// TIA Portal V20 export
// export: Created 2026-10-09T07:54:14.9470131Z, ExportSetting WithDefaults, DisplayName Totally Integrated Automation Portal, DisplayVersion V20, DisplayName TIA Portal Openness, DisplayVersion V20, DisplayName TIA Portal Teamcenter Gateway, DisplayVersion V20, DisplayName TIA Portal Version Control Interface, DisplayVersion V20, DisplayName SINAMICS Startdrive Advanced, DisplayVersion V20 SP1 Update 2, DisplayName SINAMICS Startdrive G110M, G120, G120C, G120D, G120P, G115D, DisplayVersion V20 SP1 Update 2, DisplayName SINAMICS Startdrive G130, G150, S120, S150, SINAMICS MV, G220, S200, S210, DisplayVersion V20 SP1 Update 2, DisplayName STEP 7 Professional, DisplayVersion V20, DisplayName STEP 7 Safety, DisplayVersion V20, DisplayName WinCC Basic/Comfort/Advanced, DisplayVersion V20, DisplayName WinCC Professional, DisplayVersion V20, DisplayName WinCC Unified, DisplayVersion V20
FUNCTION_BLOCK "FB_SpkAutoGraph"   // FB30, GRAPH
VERSION : 0.1
// stored: AcknowledgeErrorsRequired true, AutoNumber true, GraphVersion 6.0, InitialValuesAcquisition false, IsIECCheckEnabled false, LanguageInNetworks LAD, LockOperatingMode false, PermanentILProcessingInMANMode false, SetENOAutomatically false, SkipSteps false, UDAEnableTagReadback false, WithAlarmHandling true
   // inherited from GRAPH_BASE
   VAR
      OFF_SQ_BASE : Bool;
   END_VAR
   VAR_INPUT
      OFF_SQ { ExternalAccessible := 'False'; ExternalVisible := 'False'; ExternalWritable := 'False'} : Bool := false;   // Turn sequence off
      INIT_SQ { ExternalAccessible := 'False'; ExternalVisible := 'False'; ExternalWritable := 'False'} : Bool := false;   // Set sequence to initial state
      ACK_EF { ExternalAccessible := 'False'; ExternalVisible := 'False'; ExternalWritable := 'False'} : Bool := false;   // Acknowledge all errors and faults
      S_PREV { ExternalAccessible := 'False'; ExternalVisible := 'False'; ExternalWritable := 'False'} : Bool := false;   // Output previous step in parameter S_NO
      S_NEXT { ExternalAccessible := 'False'; ExternalVisible := 'False'; ExternalWritable := 'False'} : Bool := false;   // Indicate next step in parameter S_NO
      SW_AUTO { ExternalAccessible := 'False'; ExternalVisible := 'False'; ExternalWritable := 'False'} : Bool := false;   // Automatic mode
      SW_TAP { ExternalAccessible := 'False'; ExternalVisible := 'False'; ExternalWritable := 'False'} : Bool := false;   // Semiautomatic/switch with transition
      SW_TOP { ExternalAccessible := 'False'; ExternalVisible := 'False'; ExternalWritable := 'False'} : Bool := false;   // Semiautomatic/ignore transition
      SW_MAN { ExternalAccessible := 'False'; ExternalVisible := 'False'; ExternalWritable := 'False'} : Bool := false;   // Manual mode
      S_SEL { ExternalAccessible := 'False'; ExternalVisible := 'False'; ExternalWritable := 'False'} : Int := 0;   // Select step to be output to S_NO
      S_ON { ExternalAccessible := 'False'; ExternalVisible := 'False'; ExternalWritable := 'False'} : Bool := false;   // Activate step indicated in S_NO
      S_OFF { ExternalAccessible := 'False'; ExternalVisible := 'False'; ExternalWritable := 'False'} : Bool := false;   // Disable step indicated in S_NO
      T_PUSH { ExternalAccessible := 'False'; ExternalVisible := 'False'; ExternalWritable := 'False'} : Bool := false;   // Enable transition to switch in semi automatic mode
   END_VAR
   VAR_OUTPUT
      S_NO { ExternalAccessible := 'False'; ExternalVisible := 'False'; ExternalWritable := 'False'} : Int := 0;   // Step number
      S_MORE { ExternalAccessible := 'False'; ExternalVisible := 'False'; ExternalWritable := 'False'} : Bool := false;   // More steps are available and can be shown in S_NO
      S_ACTIVE { ExternalAccessible := 'False'; ExternalVisible := 'False'; ExternalWritable := 'False'} : Bool := false;   // Step indicated in S_NO is active
      ERR_FLT { ExternalAccessible := 'False'; ExternalVisible := 'False'; ExternalWritable := 'False'} : Bool := false;   // Interlock or supervision group error
      AUTO_ON { ExternalAccessible := 'False'; ExternalVisible := 'False'; ExternalWritable := 'False'} : Bool := false;   // Automatic mode is active
      TAP_ON { ExternalAccessible := 'False'; ExternalVisible := 'False'; ExternalWritable := 'False'} : Bool := false;   // Semiautomatic mode/step with transition enabled
      TOP_ON { ExternalAccessible := 'False'; ExternalVisible := 'False'; ExternalWritable := 'False'} : Bool := false;   // Semiautomatic mode/ignore transition enabled
      MAN_ON { ExternalAccessible := 'False'; ExternalVisible := 'False'; ExternalWritable := 'False'} : Bool := false;   // Manual mode is active
   END_VAR
   VAR_IN_OUT
      Seq : "FRK_SeqCtx";
      CylA : "FB_SpkCylinderCM";
      CylB : "FB_SpkCylinderCM";
   END_VAR
BEGIN
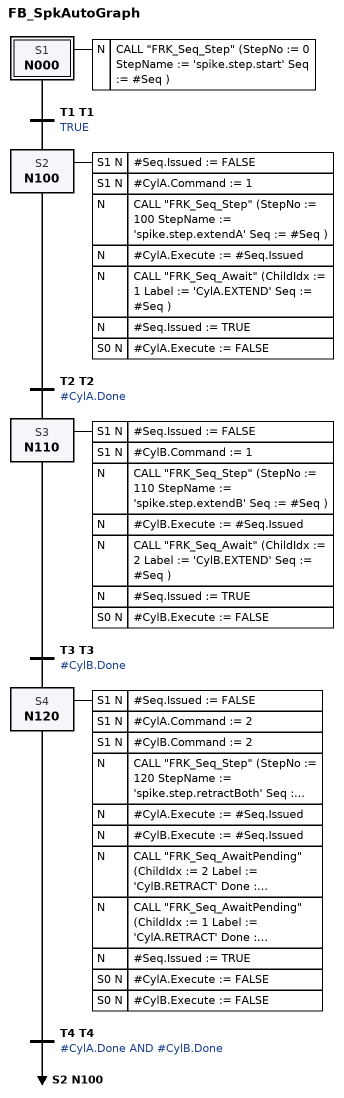
   // sequencer 1
   INITIAL_STEP N000:   // S1, max time T#10S, warning time T#7S
              N    CALL "FRK_Seq_Step" 
                   (StepNo := 0
                   StepName := 'spike.step.start'
                   Seq := #Seq
                   )
   END_STEP
   TRANSITION T1 FROM N000 TO N100   // T1
      := TRUE;
   END_TRANSITION
   STEP N100:   // S2, max time T#10S, warning time T#7S
          S1  N    #Seq.Issued := FALSE
          S1  N    #CylA.Command := 1
              N    CALL "FRK_Seq_Step" 
                   (StepNo := 100
                   StepName := 'spike.step.extendA'
                   Seq := #Seq
                   )
              N    #CylA.Execute := #Seq.Issued
              N    CALL "FRK_Seq_Await" 
                   (ChildIdx := 1
                   Label := 'CylA.EXTEND'
                   Seq := #Seq
                   )
              N    #Seq.Issued := TRUE
          S0  N    #CylA.Execute := FALSE
   END_STEP
   TRANSITION T2 FROM N100 TO N110   // T2
      := #CylA.Done;
   END_TRANSITION
   STEP N110:   // S3, max time T#10S, warning time T#7S
          S1  N    #Seq.Issued := FALSE
          S1  N    #CylB.Command := 1
              N    CALL "FRK_Seq_Step" 
                   (StepNo := 110
                   StepName := 'spike.step.extendB'
                   Seq := #Seq
                   )
              N    #CylB.Execute := #Seq.Issued
              N    CALL "FRK_Seq_Await" 
                   (ChildIdx := 2
                   Label := 'CylB.EXTEND'
                   Seq := #Seq
                   )
              N    #Seq.Issued := TRUE
          S0  N    #CylB.Execute := FALSE
   END_STEP
   TRANSITION T3 FROM N110 TO N120   // T3
      := #CylB.Done;
   END_TRANSITION
   STEP N120:   // S4, max time T#10S, warning time T#7S
          S1  N    #Seq.Issued := FALSE
          S1  N    #CylA.Command := 2
          S1  N    #CylB.Command := 2
              N    CALL "FRK_Seq_Step" 
                   (StepNo := 120
                   StepName := 'spike.step.retractBoth'
                   Seq := #Seq
                   )
              N    #CylA.Execute := #Seq.Issued
              N    #CylB.Execute := #Seq.Issued
              N    CALL "FRK_Seq_AwaitPending" 
                   (ChildIdx := 2
                   Label := 'CylB.RETRACT'
                   Done := #CylB.Done
                   Seq := #Seq
                   )
              N    CALL "FRK_Seq_AwaitPending" 
                   (ChildIdx := 1
                   Label := 'CylA.RETRACT'
                   Done := #CylA.Done
                   Seq := #Seq
                   )
              N    #Seq.Issued := TRUE
          S0  N    #CylA.Execute := FALSE
          S0  N    #CylB.Execute := FALSE
   END_STEP
   TRANSITION T4 FROM N120 TO N100   // T4, jump
      := #CylA.Done AND #CylB.Done;
   END_TRANSITION
END_FUNCTION_BLOCK
